// Test double: an access provider that also retains its table, with every store
// outcome settable, so a root's handling of a failed save or a lost table is
// tested without staging damage on the runtime's file system.
FUNCTION_BLOCK FB_ProbeAccessStore IMPLEMENTS I_AccessProvider, I_AccessStore
VAR_INPUT
    RestoreLost : BOOL;
    SaveFailed  : BOOL;
END_VAR
VAR_OUTPUT
    Serviced : UDINT;           // M_Service calls received
END_VAR

;

METHOD Authenticate : E_AccessLevel
VAR_INPUT
    User : STRING(32);
    Secret : STRING(32);
END_VAR
Authenticate := E_AccessLevel.NONE;
END_METHOD

METHOD M_Service : BOOL
Serviced := Serviced + 1;
M_Service := TRUE;
END_METHOD

METHOD M_RestoreLost : BOOL
M_RestoreLost := RestoreLost;
END_METHOD

METHOD M_SaveFailed : BOOL
M_SaveFailed := SaveFailed;
END_METHOD

END_FUNCTION_BLOCK

(* stored: Version 1.1.0.1, ProductVersion 3.1.4024.12
   POU FB_ProbeAccessStore: Id {a3f55582-6a66-4661-8a4a-0a866299ac35}, SpecialFunc None
   Method Authenticate: Id {bcfeefb1-d9e9-4b1a-a15a-b0565abcda41}
   Method M_Service: Id {0a1d3b55-5c84-4a7e-9a7b-3f1c2d4e5f61}
   Method M_RestoreLost: Id {1b2e4c66-6d95-4b8f-8b8c-4f2d3e5f6a72}
   Method M_SaveFailed: Id {2c3f5d77-7ea6-4c90-9c9d-5a3e4f6a7b83} *)
